// TIA Portal V20 export
TYPE "typeCmControlNode"
// stored: Namespace Unit1.Em6
   STRUCT
      Interlock { ExternalWritable := 'False'} : "Unit1.Em6.typeCmControlNodeInterlock";
      softcam { ExternalWritable := 'False'} : "Unit1.Em6.typeCmControlNodeSoftCam";
      brakeTest { ExternalWritable := 'False'} : "Unit1.Em6.typeCmControlNodeBrakeTest";
   END_STRUCT;
END_TYPE
